TYPE ST_AxisCtrl :
STRUCT
    Io                        :ST_AxisIo;  (*轴IO信号*)
    Status                  :ST_AxisStatus;  
    Cmd                    :ST_AxisCmd;  
END_STRUCT
END_TYPE

(* stored: Version 1.1.0.1, ProductVersion 3.1.4024.9
   DUT ST_AxisCtrl: Id {a02d953f-d359-49a0-acdf-da11fc8787f8} *)
